PROGRAM AlarmSample
VAR

END_VAR

PRG_Alarms_Core();

END_PROGRAM

(* stored: Version 1.1.0.1, ProductVersion 3.1.4024.2
   POU AlarmSample: Id {4ba2ba1f-c8f7-4c13-96f9-94d99d7108f6}, SpecialFunc None *)
